(*********************************** G.D S.p.A. - Technical Department ***********************************
============= PROGRAM INFO ============
FOLDER:             TBD
MACHINES INVOLVED:  TBD 

============= DESCRIPTION =============
csp machine declaration

============= REVISIONS ===============
Date		Version	 	Author      	Description             
----------	-------		------------  	--------------------------------------------
2019/04/05 	0000.00	 	M.Grasso		Creation of the PRG

**********************************************************************************************************)
(*$R process_ref := prc; $*)
PROGRAM csp_case_glue_os
VAR
	
	prc:											process;
	prc_path:										STRING;
	
END_VAR

_read_var_input();

_object_manager();

IF NOT objects_running()
THEN
	RETURN;	
END_IF

_read_process_image();

_mode_manager();

_set_runtime_properties();

(********************************* BODY *********************************)
(************************************************************************)

_handle_messages();

_write_output();

ACTION _handle_messages:
;
END_ACTION

ACTION _handle_process_test:
;
END_ACTION

ACTION _mode_manager:
IF process_mode_req_is_pending(prc)
THEN
    process_apply_mode_req_first_step(prc);
    CASE process_get_mode(prc) OF
        MODE_TO_ABSENT:
			;
        MODE_TO_INACTIVE:
			;
        MODE_TO_TEST:
			;
        MODE_TO_OPERATIONAL:
			;
    END_CASE
    process_apply_mode_req_second_step(prc);
END_IF
END_ACTION

ACTION _object_manager:
IF objects_initialization()
THEN
	sub_process_init(
		object_name					:= 'csp_case_glue_os.prc', 
		process						:= csp_case_glue.prc, 
		CONVERSION_this				:= prc);
		
	prc_path 						:= process_get_path(prc);
END_IF

IF objects_running()
THEN
	process_cycle(prc);
END_IF
END_ACTION

ACTION _read_process_image:
;
END_ACTION

ACTION _read_var_input:
;
END_ACTION

ACTION _set_runtime_properties:
;
END_ACTION

ACTION _write_output:
;
END_ACTION

END_PROGRAM

(* stored: Version 1.1.0.1, ProductVersion 3.1.4022.12
   POU csp_case_glue_os: Id {37e1862e-83d1-4967-bc84-91b1afa762fb}, SpecialFunc None
   Action _handle_messages: Id {abfebb4a-7fc2-46b5-8d4e-6a03f6ed5927}
   Action _handle_process_test: Id {eb651b4a-fa61-48b7-9f25-57b6ef25e20e}
   Action _mode_manager: Id {2f57c280-e0f7-45a4-9cb5-7996e376e0eb}
   Action _object_manager: Id {d057861e-9a0e-407f-9925-f12836020dea}
   Action _read_process_image: Id {b952b5ea-d2e8-41e9-92b1-7278ab4f32b4}
   Action _read_var_input: Id {5ea26260-d497-4f66-9c8f-f40f13661e6a}
   Action _set_runtime_properties: Id {7810372b-4af1-45eb-b1f3-b7dd962bf01b}
   Action _write_output: Id {594d899b-127e-4dda-bec2-3dd45e2a472c} *)
